// TIA Portal V15.1 export
// export: Created 2024-06-21T08:41:09.708933Z, ExportSetting WithDefaults, DisplayName Totally Integrated Automation Portal, DisplayVersion V15.1 Update 5, DisplayName TIA Portal Openness, DisplayVersion V15.1 Update 5, DisplayName SINAMICS Startdrive Advanced, DisplayVersion V15.1, DisplayName G130, G150, S120, S150, SINAMICS MV, S210, DisplayVersion V15.1, DisplayName G110M, G120, G120C, G120D, G120P, DisplayVersion V15.1, DisplayName STEP 7 Professional, DisplayVersion V15.1 Update 5, DisplayName STEP 7 Safety, DisplayVersion V15.1, DisplayName WinCC Professional, DisplayVersion V15.1 Update 5, DisplayName SIMATIC Visualization Architect, DisplayVersion V15.1
FUNCTION "LGBHoist2Pos2S-C-Config" : Void   // FC6646, FBD
TITLE = LMoveEPos-Config / LGBHoist2Pos2S-C-Config
{ S7_Optimized_Access := 'FALSE' }
AUTHOR : VCC
FAMILY : Config
VERSION : 0.0.0.0
// =============================================================================
// Configuration MoveUnitEpos
// =============================================================================
// =============================================================================
// Configuration of a Hoist with 2 Positions and two Speeds controlled by contactors
// =============================================================================
// stored: AutoNumber false, IsIECCheckEnabled false, SetENOAutomatically False, UDAEnableTagReadback false
   VAR_INPUT
      C_LowSpeedDetSetUsed : Bool;   // Low Speed Detection set Used
      C_LowSpeedDetResUsed : Bool;   // Low Speed Detection reset Used
      C_OverTravelSetUsed : Bool;   // Overtravel set used
      C_OverTravelResUsed : Bool;   // Overtravel reset used
      C_ContBypassOvertravelSetUsed : Bool;   // Contactor Bypass overtravel Set used
      C_ContBypassOvertravelResUsed : Bool;   // Contactor Bypass overtravel Reset used
      C_HomePosIsDown : Bool;   // The home position of the hoist is down
      C_SafetySwNc : Bool;   // Safety switch NC contact
      C_SafetySwUsed : Bool;   // Safety switch used
      C_MotorProtectionNc : Bool;   // Motor Protection NC contact
      C_MotorProtectionUsed : Bool;   // Motor Protection used
      C_EnableAlarmHW : Bool;   // Enable Alarm hardware (e.g. safetyswitch, motorprotector, detections)
      C_ReleaseBrakeUsed : Bool;   // Release brake used
      C_MotionStopUsed : Bool;   // Motion Stop used
      C_RunTimeMaxSetAlarm : DInt;   // Maximum Time (x1ms) that the function may run (create overtime) / Maximum Time (x1ms) that the function may run (create Overtime)
      C_RunTimeMaxResAlarm : DInt;   // Maximum Time (x1ms) that the function may run (create overtime) / Maximum Time (x1ms) that the function may run (create Overtime)
   END_VAR
   VAR_IN_OUT
      IO_Config : "Hoist2Pos2S-C-Config";   // Output Word / Config
   END_VAR
BEGIN

REGION Network 1: **** 1 - Inputs **** Move Bit Config
   // Move Bit Config
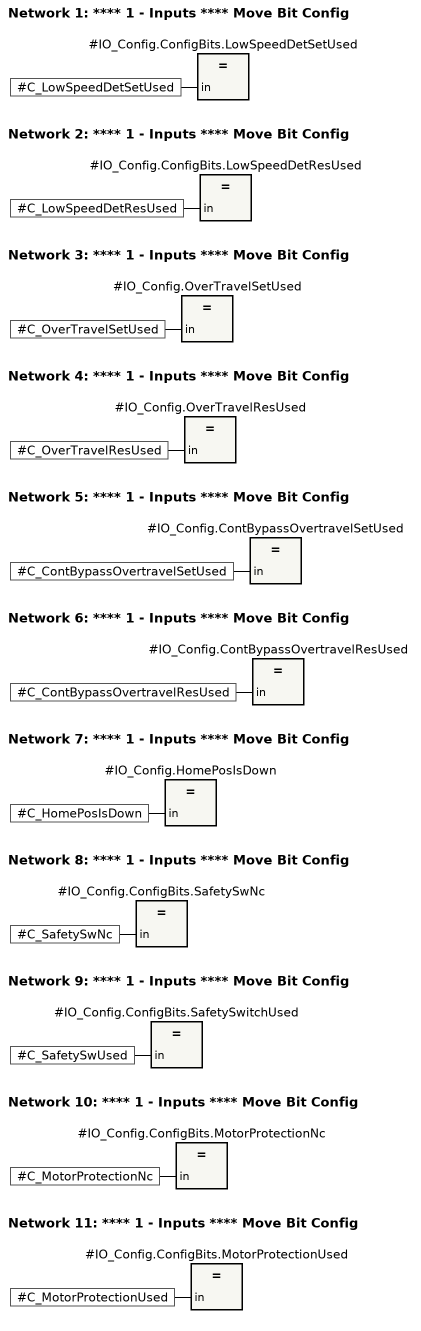
   #IO_Config.ConfigBits.LowSpeedDetSetUsed := #C_LowSpeedDetSetUsed;
END_REGION

REGION Network 2: **** 1 - Inputs **** Move Bit Config
   // Move Bit Config
   #IO_Config.ConfigBits.LowSpeedDetResUsed := #C_LowSpeedDetResUsed;
END_REGION

REGION Network 3: **** 1 - Inputs **** Move Bit Config
   #IO_Config.OverTravelSetUsed := #C_OverTravelSetUsed;
END_REGION

REGION Network 4: **** 1 - Inputs **** Move Bit Config
   #IO_Config.OverTravelResUsed := #C_OverTravelResUsed;
END_REGION

REGION Network 5: **** 1 - Inputs **** Move Bit Config
   #IO_Config.ContBypassOvertravelSetUsed := #C_ContBypassOvertravelSetUsed;
END_REGION

REGION Network 6: **** 1 - Inputs **** Move Bit Config
   #IO_Config.ContBypassOvertravelResUsed := #C_ContBypassOvertravelResUsed;
END_REGION

REGION Network 7: **** 1 - Inputs **** Move Bit Config
   #IO_Config.HomePosIsDown := #C_HomePosIsDown;
END_REGION

REGION Network 8: **** 1 - Inputs **** Move Bit Config
   // Move Bit Config
   #IO_Config.ConfigBits.SafetySwNc := #C_SafetySwNc;
END_REGION

REGION Network 9: **** 1 - Inputs **** Move Bit Config
   // Move Bit Config
   #IO_Config.ConfigBits.SafetySwitchUsed := #C_SafetySwUsed;
END_REGION

REGION Network 10: **** 1 - Inputs **** Move Bit Config
   // Move Bit Config
   #IO_Config.ConfigBits.MotorProtectionNc := #C_MotorProtectionNc;
END_REGION

REGION Network 11: **** 1 - Inputs **** Move Bit Config
   // Move Bit Config
   #IO_Config.ConfigBits.MotorProtectionUsed := #C_MotorProtectionUsed;
END_REGION

REGION Network 12: **** 1 - Inputs **** Move Bit Config
   // Move Bit Config
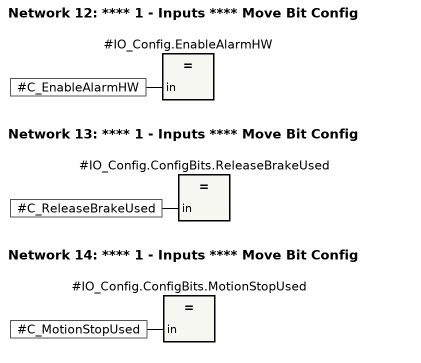
   #IO_Config.EnableAlarmHW := #C_EnableAlarmHW;
END_REGION

REGION Network 13: **** 1 - Inputs **** Move Bit Config
   // Move Bit Config
   #IO_Config.ConfigBits.ReleaseBrakeUsed := #C_ReleaseBrakeUsed;
END_REGION

REGION Network 14: **** 1 - Inputs **** Move Bit Config
   // Move Bit Config
   #IO_Config.ConfigBits.MotionStopUsed := #C_MotionStopUsed;
END_REGION

NETWORK
TITLE = **** 1 Inputs **** Move Config UDT
// Move Config
      L     #C_RunTimeMaxSetAlarm;
      T     #IO_Config.RunTimeMaxSetAlm;
      L     #C_RunTimeMaxResAlarm;
      T     #IO_Config.RunTimeMaxResAlm;
END_FUNCTION
